INTERFACE I_Lamp

// Reduces the control value by 5 in the range of 10 to 100.
METHOD DimDown
VAR_INPUT
END_VAR
END_METHOD

// Increments the control value by 5 in the range of 10 to 100.
METHOD DimUp
VAR_INPUT
END_VAR
END_METHOD

// Sets the control value to 0.
METHOD Off
VAR_INPUT
END_VAR
END_METHOD

// Sets the control value to 100.
METHOD On
VAR_INPUT
END_VAR
END_METHOD

END_INTERFACE

(* stored: Version 1.1.0.1, ProductVersion 3.1.4024.9
   Itf I_Lamp: Id {40d65e5d-c62e-4ae9-99b2-81cac6219b58}
   Method DimDown: Id {115327b1-6bf2-4c16-9a9f-a18c6ce596de}
   Method DimUp: Id {a3496324-aff1-493c-b1fe-bca8e24375de}
   Method Off: Id {41442249-3f36-4f25-8a08-dcf9ed83b1a4}
   Method On: Id {cf966bca-c883-4241-bf92-18c599ea3864} *)
